// TwinCAT 3 PLC project MainPLC
// ProgramVersion: 3.1.4024.0
// libraries:
//   Tc2_MC2, * (Beckhoff Automation GmbH)
//   Tc2_ModbusSrv, * (Beckhoff Automation GmbH)
//   Tc2_Standard, * (Beckhoff Automation GmbH)
//   Tc2_System, * (Beckhoff Automation GmbH)
//   Tc3_Module, * (Beckhoff Automation GmbH)
// project tree:
//   / GlobalTextList.TcGTLO, PlcTask.TcTTO, Visualization Manager.TcVMO (not stored)
//   GVLs/ GVL.TcGVL
//   POUs/ FB_AxisControl.TcPOU, MAIN.TcPOU, POU.TcPOU
//   VISUs/ Visualization.TcVIS
// real-time tasks:
//   TASK PlcTask: cycle T#10ms, priority 20, ADS port 350
// motion (NC):
//   TASK NC-Task 1 SAF: cycle T#2ms, priority 4, ADS port 501
//   TASK NC-Task 1 SVB: cycle T#10ms, priority 8, ADS port 511
//   AXIS Axis 1 (id 1)
//     General: UnitName=°
//     OtherSettings: AllowMotionCmdToSlave=true
//     encoder EncType=1
//     drive DrvType=5
//       Analog: TorqueSetpointScale=10, ScaleFactorActTorque=0.1
//       TimeComp: TaskDelayCycles=1
//     controller CtrType=1
//       CtrPara: PriorControlFactor=1
//         Observer: BandWidth=20

CONFIGURATION MainPLC
    RESOURCE PLC ON TwinCAT3
        TASK PlcTask(INTERVAL := T#10ms, PRIORITY := 20);
        PROGRAM MAIN WITH PlcTask : MAIN;
    END_RESOURCE
END_CONFIGURATION

// ---- GVLs/GVL.TcGVL
{attribute 'qualified_only'}
VAR_GLOBAL
	bJogForward  	: BOOL;
	bJogBackward 	: BOOL;
	{attribute 'OPC.UA.DA' := '1'}
	bEnable      	: BOOL;
	bTestBit : BOOL;
END_VAR

// ---- POUs/MAIN.TcPOU
PROGRAM MAIN
VAR

END_VAR

END_PROGRAM

// ---- POUs/FB_AxisControl.TcPOU
FUNCTION_BLOCK FB_AxisControl
VAR_INPUT
	Axis : REFERENCE TO AXIS_REF;
	MCPower : MC_Power;
	MCJog : MC_Jog;
	MCReadActVel : MC_ReadActualVelocity;
	MCReadActPos : MC_ReadActualPosition;
	bPosInterlockOK: BOOL;
	bNegInterlockOK: BOOL;
	bJogForward: BOOL;
	bJogBackward: BOOL;
	bInterlockOK: BOOL;
END_VAR
VAR_OUTPUT
END_VAR
VAR

END_VAR

MCPower(
	Axis:= Axis, 
	Enable:= bInterlockOK, 
	Enable_Positive:= bPosInterlockOK, 
	Enable_Negative:= bNegInterlockOK, 
	Override:= , 
	);
MCJog(
	Axis:= Axis, 
	JogForward:= bJogForward, 
	JogBackwards:= bJogBackward, 
	Mode:= MC_JOGMODE_STANDARD_FAST, 
	Position:= , 
	Velocity:= , 
	Acceleration:= , 
	Deceleration:= , 
	Jerk:= , 
	Done=> , 
	Busy=> , 
	Active=> , 
	CommandAborted=> , 
	Error=> , 
	ErrorID=> );
M_GetAxisData();

METHOD M_GetAxisData : BOOL
VAR_INPUT
	
END_VAR

VAR
END_VAR
MCReadActPos(
	Axis:= Axis, 
	Enable:= TRUE, 
	Valid=> , 
	Busy=> , 
	Error=> , 
	ErrorID=> , 
	Position=> );
	
MCReadActVel(
	Axis:= Axis, 
	Enable:= TRUE, 
	Valid=> , 
	Busy=> , 
	Error=> , 
	ErrorID=> , 
	ActualVelocity=> );
END_METHOD

END_FUNCTION_BLOCK

// ---- POUs/POU.TcPOU
PROGRAM POU
VAR
	btest: BOOL;
END_VAR

btest := TRUE;

END_PROGRAM

// ---- GlobalTextList.TcGTLO
TEXTLIST GlobalTextList
  970 = '%f'
  980 = 'JOG BACKWARD'
  253 = 'JOG FORWARD'
END_TEXTLIST

// ---- VISUs/Visualization.TcVIS
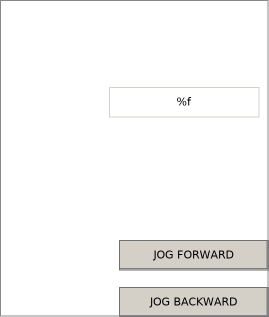
VISUALIZATION Visualization  // 269x317
    Button (119,287 150x30), "JOG BACKWARD"
        tap GVL.bJogBackward
    Button (119,240 150x30), "JOG FORWARD"
        tap GVL.bJogForward
    Textfield (109,87 150x30), "%f", text variable: MAIN.AxisControlConv1.fbMCReadActPos.Position
END_VISUALIZATION
